(* PLC project Controller, Unknown Controller 1 *)
(* stored: creationDateTime 2022-08-16T15:49:17, modificationDateTime 2023-12-28T19:43:36 *)

PROGRAM pump
  VAR_EXTERNAL
    humidity_set_point : REAL;
    humidity : REAL;
  END_VAR
  VAR
    hist : REAL := 5.0;
  END_VAR
  VAR_EXTERNAL
    pump_state : BOOL;
  END_VAR
  VAR
    HYSTERESIS0 : HYSTERESIS;
    TON0 : TON;
    TON_TIME : TIME;
    TON1 : TON;
    RS0 : RS;
  END_VAR
  VAR_EXTERNAL
    relay_access : BOOL;
  END_VAR
  VAR  (* added by the conversion: wires and edge detectors of the diagram *)
    _AND51_OUT : BOOL;
  END_VAR

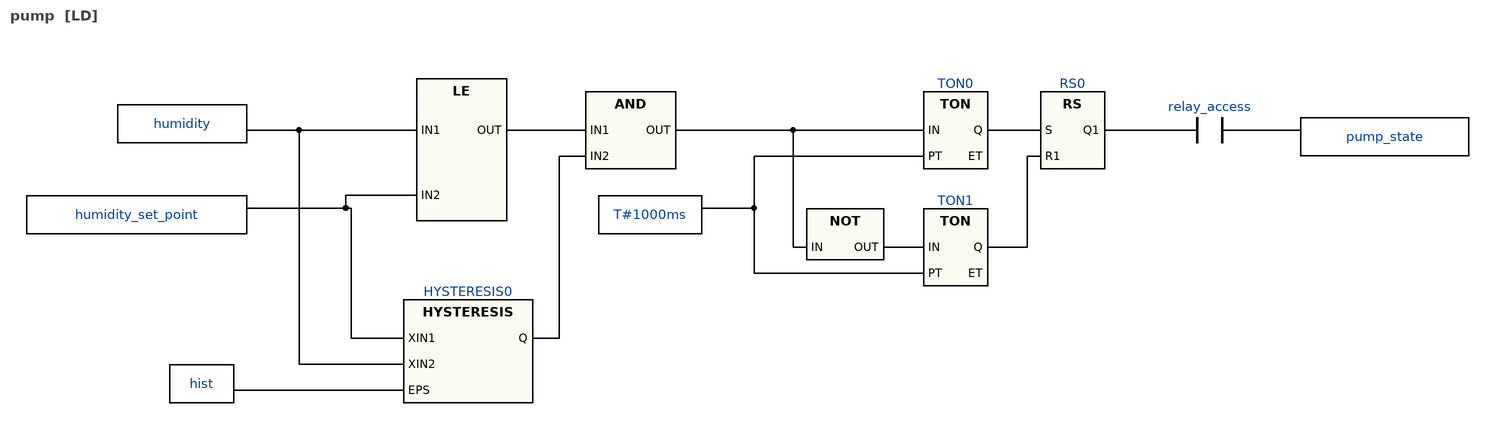
(* LD diagram, written out as Structured Text *)
HYSTERESIS0(XIN1 := humidity_set_point, XIN2 := humidity, EPS := hist);
_AND51_OUT := humidity <= humidity_set_point AND HYSTERESIS0.Q;
TON0(IN := _AND51_OUT, PT := T#1000ms);
TON1(IN := NOT _AND51_OUT, PT := T#1000ms);
RS0(S := TON0.Q, R1 := TON1.Q);
pump_state := RS0.Q1 AND relay_access;
END_PROGRAM

PROGRAM heater
  VAR_EXTERNAL
    temp_set_point : REAL;
  END_VAR
  VAR
    hist : REAL := 5.0;
  END_VAR
  VAR_EXTERNAL
    temperature : REAL;
    heater_state : BOOL;
  END_VAR
  VAR
    HYSTERESIS0 : HYSTERESIS;
    TON0 : TON;
    TON_TIME : TIME;
    TON1 : TON;
    RS0 : RS;
  END_VAR
  VAR_EXTERNAL
    relay_access : BOOL;
  END_VAR
  VAR  (* added by the conversion: wires and edge detectors of the diagram *)
    _AND51_OUT : BOOL;
  END_VAR

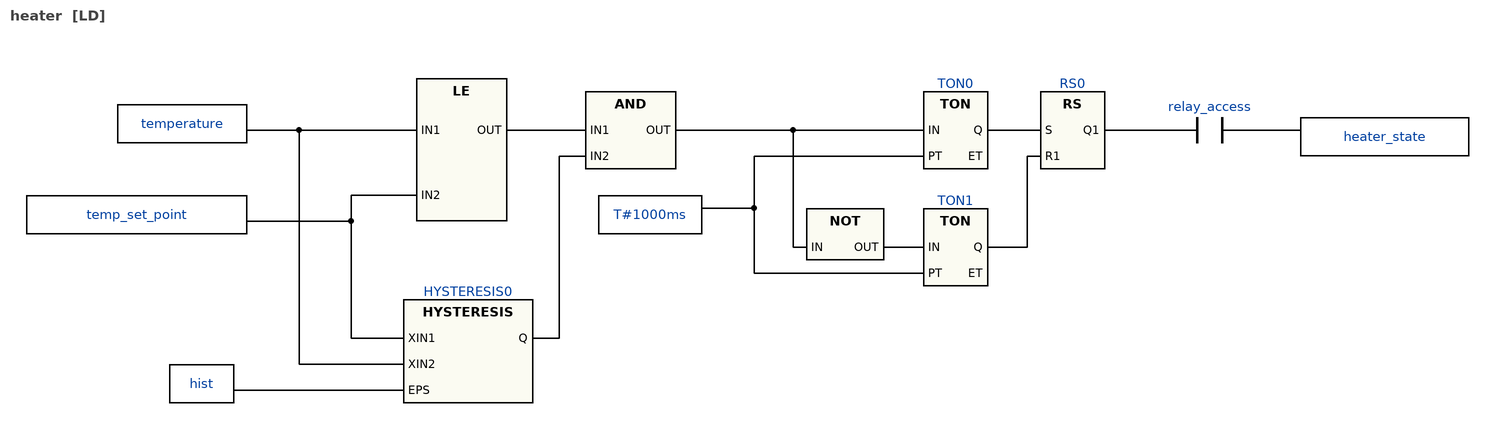
(* LD diagram, written out as Structured Text *)
HYSTERESIS0(XIN1 := temp_set_point, XIN2 := temperature, EPS := hist);
_AND51_OUT := temperature <= temp_set_point AND HYSTERESIS0.Q;
TON0(IN := _AND51_OUT, PT := T#1000ms);
TON1(IN := NOT _AND51_OUT, PT := T#1000ms);
RS0(S := TON0.Q, R1 := TON1.Q);
heater_state := RS0.Q1 AND relay_access;
END_PROGRAM

PROGRAM temp
  VAR
    ADC_IN_0 AT %IW0 : UINT := 0;
  END_VAR
  VAR
    CONST_1_REAL : REAL := 1.0;
    CONST_10_REAL : REAL := 10.0;
    ADC_MAX_VAL : REAL := 65535.0;
    CONST_KELVIN : REAL := 273.15;
    CONST_RES_DIV : REAL := 100000.0;
    CONST_RES_NTC : REAL := 10000.0;
    CONST_BETA : REAL := 3200.0;
    CONST_1_DIV_T0 : REAL := 0.003355;
  END_VAR
  VAR_EXTERNAL
    ntc_resistance : REAL;
    temperature : REAL;
  END_VAR
  VAR  (* added by the conversion: wires and edge detectors of the diagram *)
    _DIV20_OUT : REAL;
  END_VAR

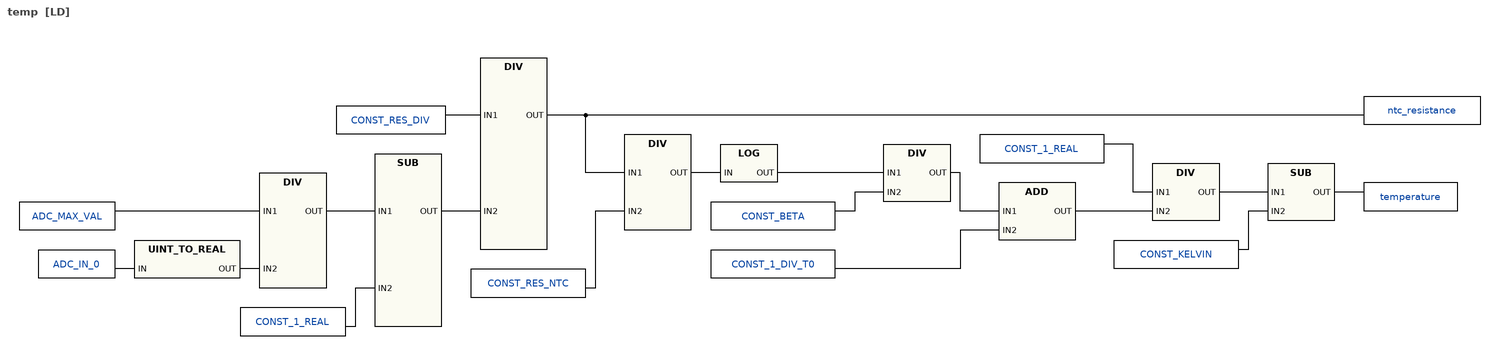
(* LD diagram, written out as Structured Text *)
_DIV20_OUT := CONST_RES_DIV / (ADC_MAX_VAL / UINT_TO_REAL(ADC_IN_0) - CONST_1_REAL);
ntc_resistance := _DIV20_OUT;
temperature := CONST_1_REAL / (LOG(_DIV20_OUT / CONST_RES_NTC) / CONST_BETA + CONST_1_DIV_T0) - CONST_KELVIN;
END_PROGRAM

PROGRAM mqtt
  VAR
    TON0 : TON;
    TOF0 : TOF;
    MQTT_SEND0 : MQTT_SEND;
    MQTT_SEND1 : MQTT_SEND;
    MQTT_SEND2 : MQTT_SEND;
    MQTT_SEND3 : MQTT_SEND;
    MQTT_CONNECT0 : MQTT_CONNECT;
    PUBLISH_CYCLE : TIME := T#5000ms;
    trigger_send : BOOL;
    trigger_receive : BOOL := FALSE;
    trigger_receive_hum : BOOL := FALSE;
    mqtt_connected : BOOL;
  END_VAR
  VAR_EXTERNAL
    temperature : REAL;
    humidity : REAL;
    ntc_resistance : REAL;
    temp_set_point : REAL;
    humidity_set_point : REAL;
    heater_state : BOOL;
    pump_state : BOOL;
  END_VAR
  VAR
    MQTT_SUBSCRIBE0 : MQTT_SUBSCRIBE;
    MQTT_RECEIVE0 : MQTT_RECEIVE;
    MQTT_SEND4 : MQTT_SEND;
    MQTT_SEND5 : MQTT_SEND;
    MQTT_SUBSCRIBE1 : MQTT_SUBSCRIBE;
    MQTT_RECEIVE1 : MQTT_RECEIVE;
  END_VAR

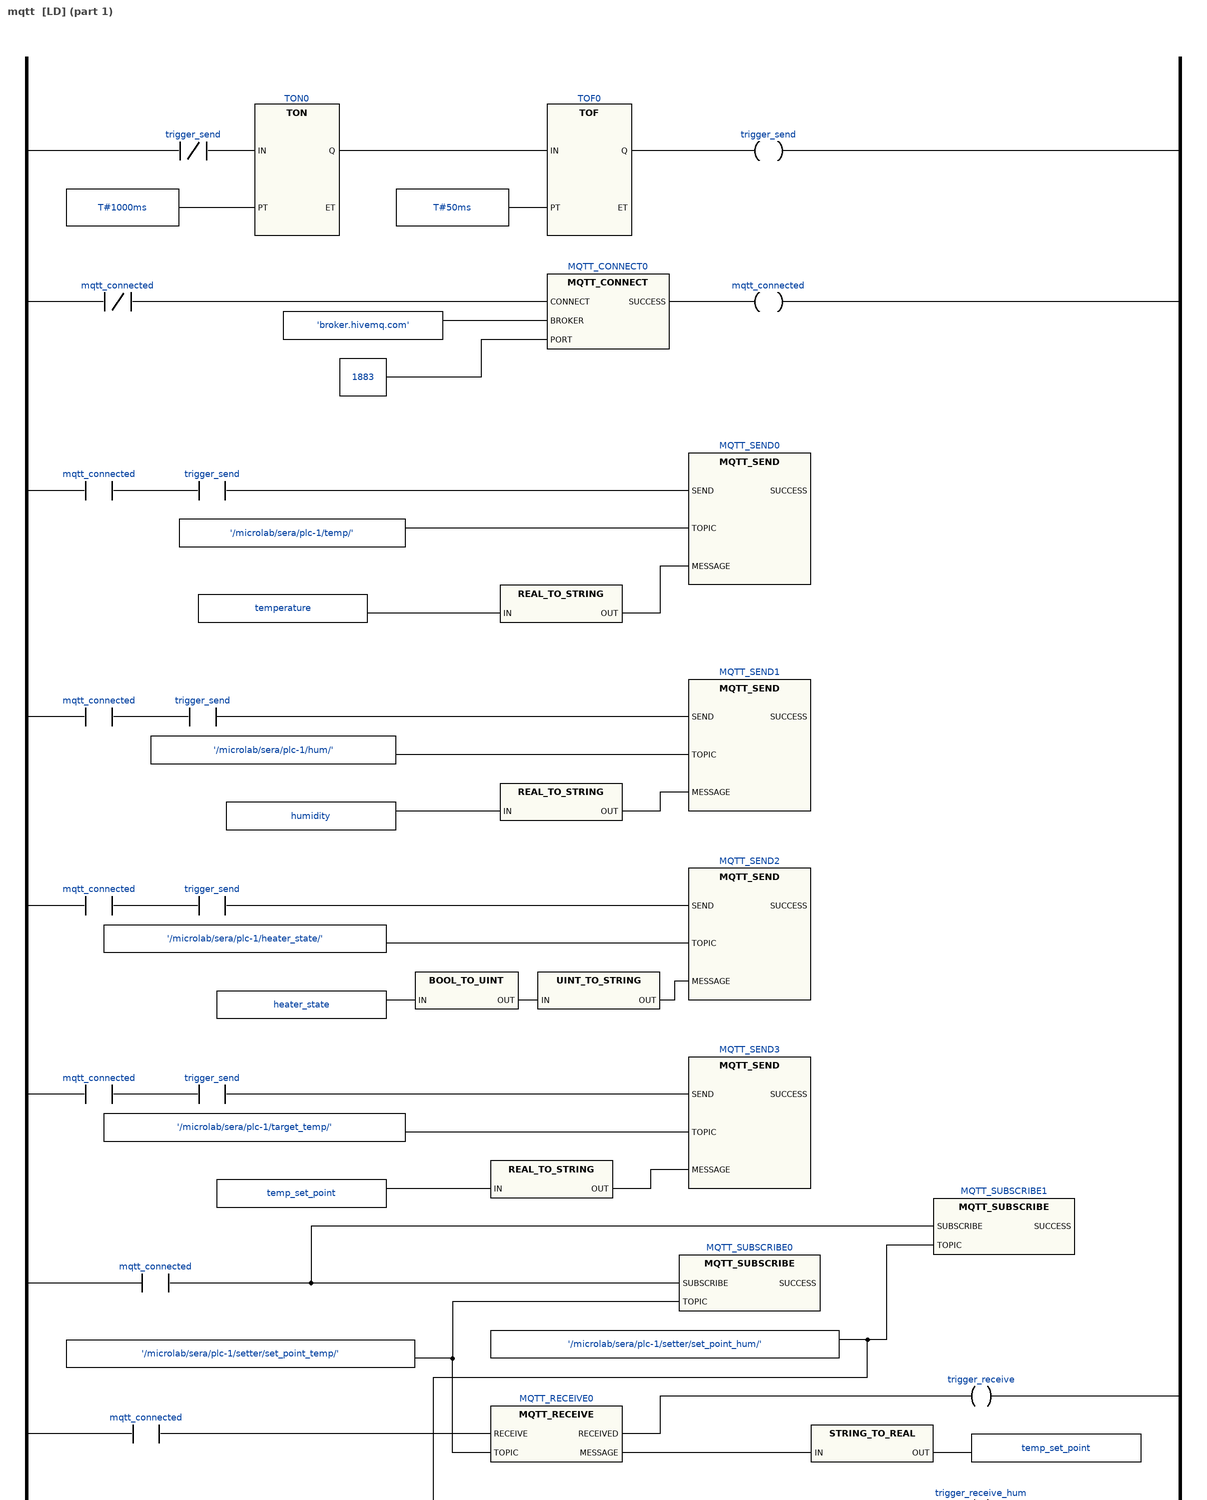
(* LD diagram, written out as Structured Text *)
TON0(IN := NOT trigger_send, PT := T#1000ms);
TOF0(IN := TON0.Q, PT := T#50ms);
trigger_send := TOF0.Q;
MQTT_CONNECT0(CONNECT := NOT mqtt_connected, BROKER := 'broker.hivemq.com', PORT := 1883);
mqtt_connected := MQTT_CONNECT0.SUCCESS;
MQTT_RECEIVE0(RECEIVE := mqtt_connected, TOPIC := '/microlab/sera/plc-1/setter/set_point_temp/');
trigger_receive := MQTT_RECEIVE0.RECEIVED;
temp_set_point := STRING_TO_REAL(MQTT_RECEIVE0.MESSAGE);
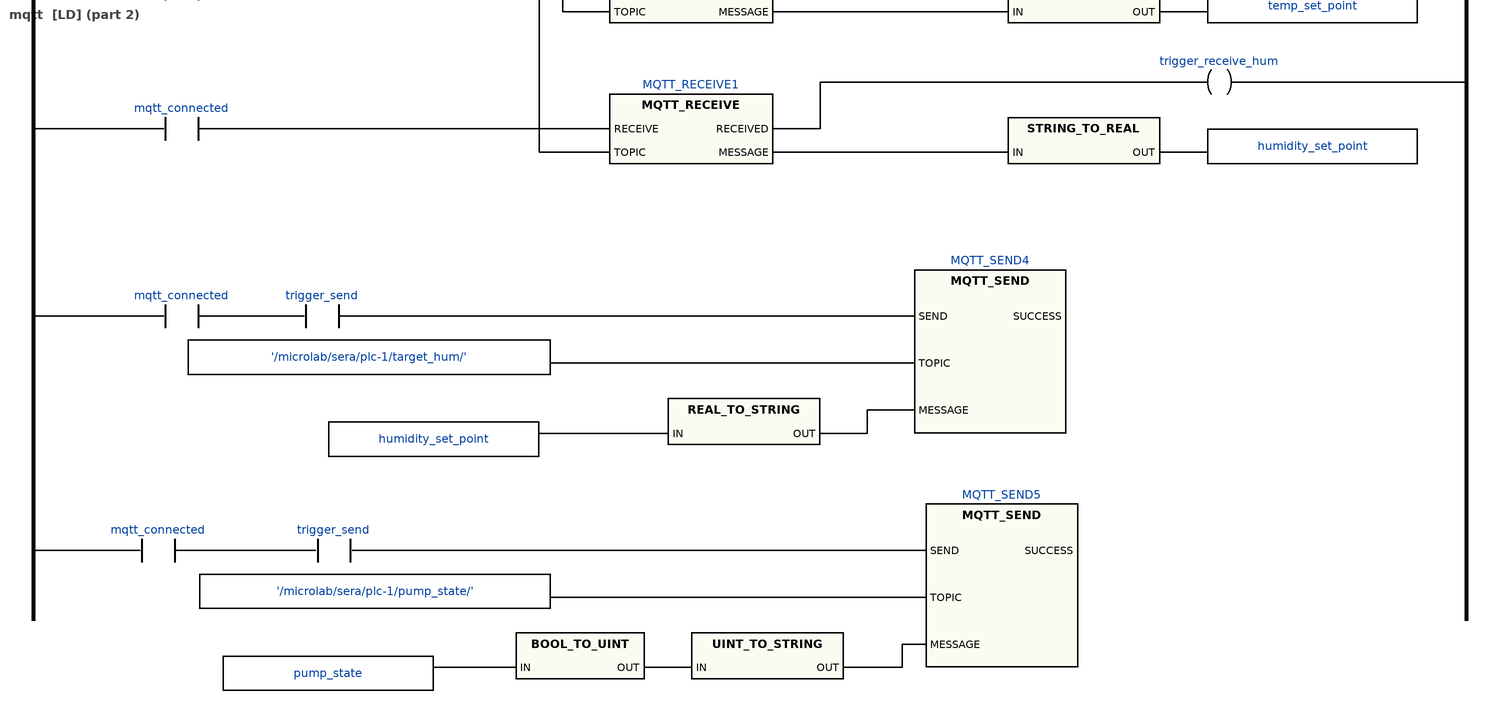
MQTT_RECEIVE1(RECEIVE := mqtt_connected, TOPIC := '/microlab/sera/plc-1/setter/set_point_hum/');
trigger_receive_hum := MQTT_RECEIVE1.RECEIVED;
humidity_set_point := STRING_TO_REAL(MQTT_RECEIVE1.MESSAGE);
MQTT_SEND0(SEND := mqtt_connected AND trigger_send, TOPIC := '/microlab/sera/plc-1/temp/', MESSAGE := REAL_TO_STRING(temperature));
MQTT_SEND1(SEND := mqtt_connected AND trigger_send, TOPIC := '/microlab/sera/plc-1/hum/', MESSAGE := REAL_TO_STRING(humidity));
MQTT_SEND2(SEND := mqtt_connected AND trigger_send, TOPIC := '/microlab/sera/plc-1/heater_state/', MESSAGE := UINT_TO_STRING(BOOL_TO_UINT(heater_state)));
MQTT_SEND3(SEND := mqtt_connected AND trigger_send, TOPIC := '/microlab/sera/plc-1/target_temp/', MESSAGE := REAL_TO_STRING(temp_set_point));
MQTT_SUBSCRIBE1(SUBSCRIBE := mqtt_connected, TOPIC := '/microlab/sera/plc-1/setter/set_point_hum/');
MQTT_SUBSCRIBE0(SUBSCRIBE := mqtt_connected, TOPIC := '/microlab/sera/plc-1/setter/set_point_temp/');
MQTT_SEND4(SEND := mqtt_connected AND trigger_send, TOPIC := '/microlab/sera/plc-1/target_hum/', MESSAGE := REAL_TO_STRING(humidity_set_point));
MQTT_SEND5(SEND := mqtt_connected AND trigger_send, TOPIC := '/microlab/sera/plc-1/pump_state/', MESSAGE := UINT_TO_STRING(BOOL_TO_UINT(pump_state)));
END_PROGRAM

PROGRAM main
  VAR
    ADC_OUT_1 AT %QW0 : UINT := 5000;
    button_verde_start AT %IX0.0 : BOOL := FALSE;
    button_rosu_stop AT %IX0.1 : BOOL := FALSE;
  END_VAR
  VAR_EXTERNAL
    relay_access : BOOL;
  END_VAR
  VAR
    ADC_IN_1 AT %IW1 : UINT := 0;
  END_VAR
  VAR_EXTERNAL
    humidity : REAL;
  END_VAR

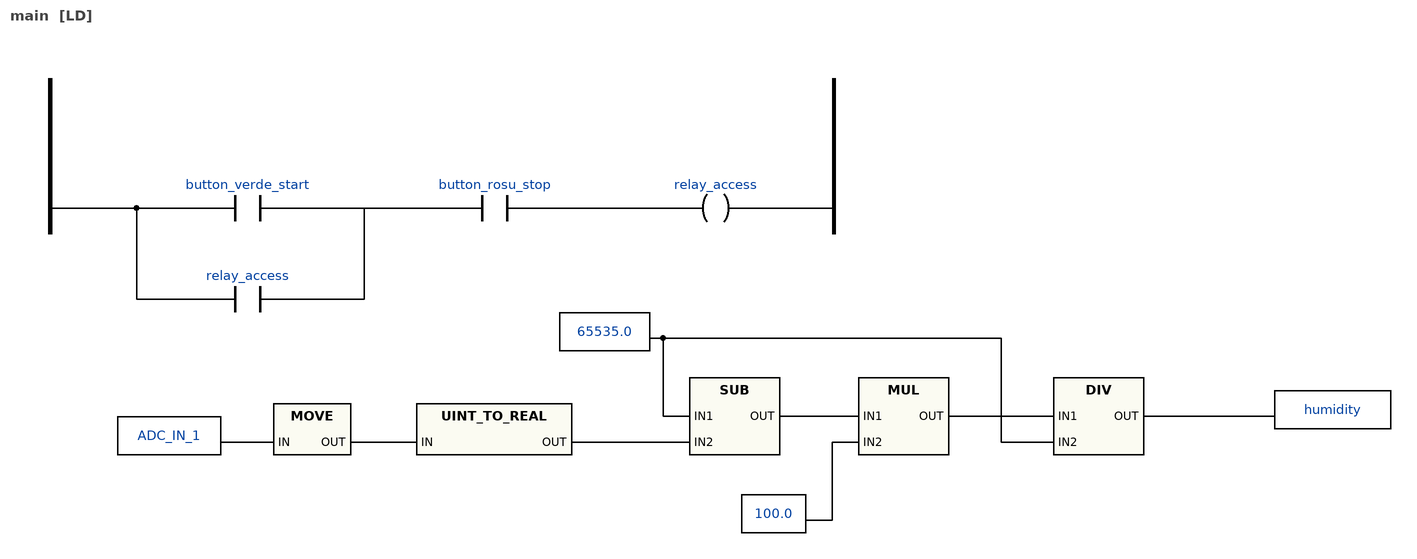
(* LD diagram, written out as Structured Text *)
relay_access := (button_verde_start OR relay_access) AND button_rosu_stop;
humidity := (65535.0 - UINT_TO_REAL(ADC_IN_1)) * 100.0 / 65535.0;
END_PROGRAM

CONFIGURATION Config0
  RESOURCE Res0 ON PLC
    VAR_GLOBAL
      temp_set_point : REAL := 18.0;
      temperature : REAL := 0.0;
      humidity_set_point : REAL := 25;
      humidity : REAL := 0.0;
      ntc_resistance : REAL := 0.0;
      relay_access : BOOL := FALSE;
      heater_state AT %QX0.0 : BOOL := FALSE;
      pump_state AT %QX0.1 : BOOL := FALSE;
    END_VAR
    TASK task0(INTERVAL := T#50ms, PRIORITY := 0);
    TASK task1(INTERVAL := T#20ms, PRIORITY := 0);
    TASK task2(INTERVAL := T#100ms, PRIORITY := 0);
    PROGRAM instance0 WITH task0 : main;
    PROGRAM instance2 WITH task0 : temp;
    PROGRAM instance1 WITH task1 : mqtt;
    PROGRAM instance3 WITH task2 : heater;
    PROGRAM instance4 WITH task2 : pump;
  END_RESOURCE
END_CONFIGURATION
